// ___EM_Instance_9

// EM Instance DB
// EM_Instance_9
// DB726 = EM_Instance_9
// FB702 = EM_I_OUT
DATA_BLOCK DB726 FB702
BEGIN
END_DATA_BLOCK

FUNCTION "EM_Instance_9_FC" : VOID
TITLE =EM_Instance_9_FC
// EM_Instance_9_FC

AUTHOR :
FAMILY : 'eminst'
NAME : namehead
VERSION : 0.1

BEGIN

NETWORK
TITLE = Main
//--------------------------------
//
//--------------------------------

CALL EM_I_OUT, DB 726(
	em_id := 34,
	Pump_RUN := "M106".QNOFF2,
	PIC01_PV := "FIC101".PV,
	LT01_PV := "LT200".QfVal,
	BV_Bottom_OPN := "MV007".QOPEN,
	BV_Bottom_CLS := "MV007".QCLOSE,
	BV_Tran_M04_OPN := "MV003".QOPEN,
	BV_Tran_M04_CLS := "MV003".QCLOSE,
	Pump_ON := "M106".L_ON,
	PIC01_SP := "FIC101".HMI_SP_INT,
	PIC01_AUT := "FIC101".L_AUT,
	PIC01_VAL_OUT := "FIC101".HMI_MAN,
	PIC01_SET_SP := "FIC101".Set_SP,
	PIC01_SET_OUT := "FIC101".Set_Output,
	BV_Bottom_CMD := "MV007".AUT_OP,
	BV_Tran_M04_CMD := "MV003".AUT_OP
)



END_FUNCTION


// <SPLIT>EM_INSTANCE_EM_Instance_10.awl</SPLIT>


// ___EM_Instance_10

// EM Instance DB
// EM_Instance_10
// DB727 = EM_Instance_10
// FB702 = EM_I_OUT
DATA_BLOCK DB727 FB702
BEGIN
END_DATA_BLOCK

FUNCTION "EM_Instance_10_FC" : VOID
TITLE =EM_Instance_10_FC
// EM_Instance_10_FC

AUTHOR :
FAMILY : 'eminst'
NAME : namehead
VERSION : 0.1

BEGIN

NETWORK
TITLE = Main
//--------------------------------
//
//--------------------------------

CALL EM_I_OUT, DB 727(
	em_id := 35,
	Pump_RUN := "M106".QNOFF2,
	PIC01_PV := "FIC101".PV,
	LT01_PV := "LT101".QfVal,
	BV_Bottom_OPN := "MV007".QOPEN,
	BV_Bottom_CLS := "MV007".QCLOSE,
	Pump_ON := "M106".L_ON,
	PIC01_SP := "FIC101".HMI_SP_INT,
	PIC01_AUT := "FIC101".L_AUT,
	PIC01_VAL_OUT := "FIC101".HMI_MAN,
	PIC01_SET_SP := "FIC101".Set_SP,
	PIC01_SET_OUT := "FIC101".Set_Output,
	BV_Bottom_CMD := "MV007".AUT_OP
)



END_FUNCTION


// <SPLIT>EM_INSTANCE_EM_Instance_11.awl</SPLIT>


// ___EM_Instance_11

// EM Instance DB
// EM_Instance_11
// DB728 = EM_Instance_11
// FB702 = EM_I_OUT
DATA_BLOCK DB728 FB702
BEGIN
END_DATA_BLOCK

FUNCTION "EM_Instance_11_FC" : VOID
TITLE =EM_Instance_11_FC
// EM_Instance_11_FC

AUTHOR :
FAMILY : 'eminst'
NAME : namehead
VERSION : 0.1

BEGIN

NETWORK
TITLE = Main
//--------------------------------
//
//--------------------------------

CALL EM_I_OUT, DB 728(
	em_id := 36,
	Pump_RUN := "M106".QNOFF2,
	PIC01_PV := "FIC101".PV,
	LT01_PV := "LT201".QfVal,
	XV_Bottom_OPN := "XV001".QOPEN,
	XV_Bottom_CLS := "XV001".QCLOSE,
	Pump_ON := "M106".L_ON,
	PIC01_SP := "FIC101".HMI_SP_INT,
	PIC01_AUT := "FIC101".L_AUT,
	PIC01_VAL_OUT := "FIC101".HMI_MAN,
	PIC01_SET_SP := "FIC101".Set_SP,
	PIC01_SET_OUT := "FIC101".Set_Output,
	XV_Bottom_CMD := "XV001".AUT_OP
)



END_FUNCTION


// <SPLIT>EM_INSTANCE_EM_Instance_12.awl</SPLIT>


// ___EM_Instance_12

// EM Instance DB
// EM_Instance_12
// DB729 = EM_Instance_12
// FB702 = EM_I_OUT
DATA_BLOCK DB729 FB702
BEGIN
END_DATA_BLOCK

FUNCTION "EM_Instance_12_FC" : VOID
TITLE =EM_Instance_12_FC
// EM_Instance_12_FC

AUTHOR :
FAMILY : 'eminst'
NAME : namehead
VERSION : 0.1

BEGIN

NETWORK
TITLE = Main
//--------------------------------
//
//--------------------------------

CALL EM_I_OUT, DB 729(
	em_id := 37,
	Pump_RUN := "M106".QNOFF2,
	PIC01_PV := "FIC101".PV,
	LT01_PV := "LT201".QfVal,
	XV_Bottom_OPN := "XV002".QOPEN,
	XV_Bottom_CLS := "XV002".QCLOSE,
	Pump_ON := "M106".L_ON,
	PIC01_SP := "FIC101".HMI_SP_INT,
	PIC01_AUT := "FIC101".L_AUT,
	PIC01_VAL_OUT := "FIC101".HMI_MAN,
	PIC01_SET_SP := "FIC101".Set_SP,
	PIC01_SET_OUT := "FIC101".Set_Output,
	XV_Bottom_CMD := "XV002".AUT_OP
)



END_FUNCTION


// <SPLIT>EM_INSTANCE_EM_Instance_13.awl</SPLIT>


// ___EM_Instance_13

// EM Instance DB
// EM_Instance_13
// DB730 = EM_Instance_13
// FB702 = EM_I_OUT
DATA_BLOCK DB730 FB702
BEGIN
END_DATA_BLOCK

FUNCTION "EM_Instance_13_FC" : VOID
TITLE =EM_Instance_13_FC
// EM_Instance_13_FC

AUTHOR :
FAMILY : 'eminst'
NAME : namehead
VERSION : 0.1

BEGIN

NETWORK
TITLE = Main
//--------------------------------
//
//--------------------------------

CALL EM_I_OUT, DB 730(
	em_id := 38,
	Pump_RUN := "M106".QNOFF2,
	PIC01_PV := "FIC101".PV,
	LT01_PV := "LT201".QfVal,
	XV_Bottom_OPN := "XV003".QOPEN,
	XV_Bottom_CLS := "XV003".QCLOSE,
	Pump_ON := "M106".L_ON,
	PIC01_SP := "FIC101".HMI_SP_INT,
	PIC01_AUT := "FIC101".L_AUT,
	PIC01_VAL_OUT := "FIC101".HMI_MAN,
	PIC01_SET_SP := "FIC101".Set_SP,
	PIC01_SET_OUT := "FIC101".Set_Output,
	XV_Bottom_CMD := "XV003".AUT_OP
)



END_FUNCTION


// <SPLIT>EM_INSTANCE_EM_Instance_14.awl</SPLIT>


// ___EM_Instance_14

// EM Instance DB
// EM_Instance_14
// DB731 = EM_Instance_14
// FB702 = EM_I_OUT
DATA_BLOCK DB731 FB702
BEGIN
END_DATA_BLOCK

FUNCTION "EM_Instance_14_FC" : VOID
TITLE =EM_Instance_14_FC
// EM_Instance_14_FC

AUTHOR :
FAMILY : 'eminst'
NAME : namehead
VERSION : 0.1

BEGIN

NETWORK
TITLE = Main
//--------------------------------
//
//--------------------------------

CALL EM_I_OUT, DB 731(
	em_id := 39,
	Pump_RUN := "M106".QNOFF2,
	PIC01_PV := "FIC101".PV,
	LT01_PV := "LT201".QfVal,
	XV_Bottom_OPN := "XV004".QOPEN,
	XV_Bottom_CLS := "XV004".QCLOSE,
	Pump_ON := "M106".L_ON,
	PIC01_SP := "FIC101".HMI_SP_INT,
	PIC01_AUT := "FIC101".L_AUT,
	PIC01_VAL_OUT := "FIC101".HMI_MAN,
	PIC01_SET_SP := "FIC101".Set_SP,
	PIC01_SET_OUT := "FIC101".Set_Output,
	XV_Bottom_CMD := "XV004".AUT_OP
)



END_FUNCTION



// <SPLIT>PHASE_INSTANCE_phase_1.awl</SPLIT>


// ___phase_1

// Phase Instance DB
// DB716 = phase_1
// FB701 = phase_example
DATA_BLOCK DB716 FB701
BEGIN
END_DATA_BLOCK

FUNCTION "phase_1_FC" : VOID
TITLE =phase_1_FC
// phase_1_FC
// First instance of fds_example
AUTHOR :
FAMILY : 'phseinst'
NAME : namehead
VERSION : 0.1

BEGIN
NETWORK
TITLE = Main
//--------------------------------
// Call the phase
//--------------------------------

CALL phase_example, DB 716
	(XV003_OPN := "XV300".QOPEN,
	XV004_OPN := "XV400".QOPEN,
	XV005_OPN := "XV500".QOPEN,
	P001_RUN := "P100".QRUN,
	LT001_PV := "LT100".QfVal,
	LT002_PV := "LT200".QfVal,
	XV003_CMD := "XV300".AUT_OP,
	XV004_CMD := "XV400".AUT_OP,
	P001_ON := "P100".AUTO_ON,
	FIC001_EXT := "FIC100".L_REMOTE,
	FIC001_SP := "FIC100".HMI_SP_INT,
	FIC001_AUT := "FIC100".L_AUT,
	FIC001_VAL_OUT := "FIC100".HMI_MAN,
	FIC001_SET_SP := "FIC100".Set_SP,
	FIC001_SET_OUT := "FIC100".Set_Output);



END_FUNCTION


// <SPLIT>PHASE_INSTANCE_phase_2.awl</SPLIT>


// ___phase_2

// Phase Instance DB
// DB717 = phase_2
// FB701 = phase_example
DATA_BLOCK DB717 FB701
BEGIN
END_DATA_BLOCK

FUNCTION "phase_2_FC" : VOID
TITLE =phase_2_FC
// phase_2_FC
// Second instance of fds_example
AUTHOR :
FAMILY : 'phseinst'
NAME : namehead
VERSION : 0.1

BEGIN
NETWORK
TITLE = Main
//--------------------------------
// Call the phase
//--------------------------------

CALL phase_example, DB 717
	(XV003_OPN := "XV301".QOPEN,
	XV004_OPN := "XV401".QOPEN,
	XV005_OPN := "XV501".QOPEN,
	P001_RUN := "P101".QRUN,
	LT001_PV := "LT101".QfVal,
	LT002_PV := "LT201".QfVal,
	XV003_CMD := "XV301".AUT_OP,
	XV004_CMD := "XV401".AUT_OP,
	P001_ON := "P101".AUTO_ON,
	FIC001_EXT := "FIC101".L_REMOTE,
	FIC001_SP := "FIC101".HMI_SP_INT,
	FIC001_AUT := "FIC101".L_AUT,
	FIC001_VAL_OUT := "FIC101".HMI_MAN,
	FIC001_SET_SP := "FIC101".Set_SP,
	FIC001_SET_OUT := "FIC101".Set_Output);



END_FUNCTION


// <SPLIT>main_program.awl</SPLIT>

// ___Control_Modules
FUNCTION Control_Modules : VOID
TITLE = Control_Modules
// Call all the Control Modules
AUTHOR:
FAMILY: 'program'
NAME: namehead
VERSION: 0.1

BEGIN

NETWORK
TITLE =
//--------------------------------
//
//--------------------------------
	CALL	XV001_FC;
	CALL	XV002_FC;
	CALL	XV003_FC;
	CALL	XV004_FC;
	CALL	XV300_FC;
	CALL	XV400_FC;
	CALL	XV500_FC;
	CALL	XV301_FC;
	CALL	XV501_FC;
	CALL	XV401_FC;
	CALL	MV001_FC;
	CALL	MV002_FC;
	CALL	MV003_FC;
	CALL	MV004_FC;
	CALL	MV005_FC;
	CALL	MV006_FC;
	CALL	MV007_FC;
	CALL	P100_FC;
	CALL	P200_FC;
	CALL	P101_FC;
	CALL	P201_FC;
	CALL	M100_FC;
	CALL	M101_FC;
	CALL	M102_FC;
	CALL	M103_FC;
	CALL	M104_FC;
	CALL	M105_FC;
	CALL	M106_FC;
	CALL	LT001_FC;
	CALL	LT002_FC;
	CALL	LT003_FC;
	CALL	LT004_FC;
	CALL	LT005_FC;
	CALL	LT006_FC;
	CALL	LT007_FC;
	CALL	LT100_FC;
	CALL	LT200_FC;
	CALL	LT101_FC;
	CALL	LT201_FC;
	CALL	LS001_FC;
	CALL	LS002_FC;
	CALL	LIC001_FC;
	CALL	LIC002_FC;
	CALL	LIC003_FC;
	CALL	LIC004_FC;
	CALL	LIC005_FC;
	CALL	LIC006_FC;
	CALL	FIC100_FC;
	CALL	FIC101_FC;

END_FUNCTION

// ___Equipment_Modules
FUNCTION Equipment_Modules : VOID
TITLE = Equipment_Modules
// Call all the Equipment Modules
AUTHOR:
FAMILY: 'program'
NAME: namehead
VERSION: 0.1

BEGIN

NETWORK
TITLE =
//--------------------------------
//
//--------------------------------
	CALL	EM_Instance_1_FC;
	CALL	EM_Instance_2_FC;
	CALL	EM_Instance_3_FC;
	CALL	EM_Instance_4_FC;
	CALL	EM_Instance_5_FC;
	CALL	EM_Instance_6_FC;
	CALL	EM_Instance_7_FC;
	CALL	EM_Instance_8_FC;
	CALL	EM_Instance_9_FC;
	CALL	EM_Instance_10_FC;
	CALL	EM_Instance_11_FC;
	CALL	EM_Instance_12_FC;
	CALL	EM_Instance_13_FC;
	CALL	EM_Instance_14_FC;

END_FUNCTION

// ___Phases
FUNCTION Phases : VOID
TITLE = Phases
// Call all the Phases
AUTHOR:
FAMILY: 'program'
NAME: namehead
VERSION: 0.1

BEGIN

NETWORK
TITLE =
//--------------------------------
//
//--------------------------------
	CALL	phase_1_FC;
	CALL	phase_2_FC;

END_FUNCTION

// ___Units
FUNCTION Units : VOID
TITLE = Units
// Call all the Units
AUTHOR:
FAMILY: 'program'
NAME: namehead
VERSION: 0.1

BEGIN

NETWORK
TITLE =
//--------------------------------
//
//--------------------------------

END_FUNCTION

// ___Main_Program
FUNCTION Main_Program : VOID
TITLE = Main_Program
// Call all the program components
AUTHOR:
FAMILY: 'program'
NAME: namehead
VERSION: 0.1

BEGIN

NETWORK
TITLE =
//--------------------------------
//
//--------------------------------

	CALL	Control_Modules;
	CALL	Equipment_Modules;
	CALL	Phases;
	CALL	Units;

END_FUNCTION

// ___OB1
// OB1 only calls Main_Program
// Comment this whole section if some code needs to be entered manually
// => in this case make another program structure starting from OB1
ORGANIZATION_BLOCK OB 1
TITLE = "Main Program Sweep (Cycle)"
VERSION : 0.1


VAR_TEMP
  OB1_EV_CLASS : BYTE ;	//Bits 0-3 = 1 (Coming event), Bits 4-7 = 1 (Event class 1)
  OB1_SCAN_1 : BYTE ;	//1 (Cold restart scan 1 of OB 1), 3 (Scan 2-n of OB 1)
  OB1_PRIORITY : BYTE ;	//Priority of OB Execution
  OB1_OB_NUMBR : BYTE ;	//1 (Organization block 1, OB1)
  OB1_RESERVED_1 : BYTE ;	//Reserved for system
  OB1_RESERVED_2 : BYTE ;	//Reserved for system
  OB1_PREV_CYCLE : INT ;	//Cycle time of previous OB1 scan (milliseconds)
  OB1_MIN_CYCLE : INT ;	//Minimum cycle time of OB1 (milliseconds)
  OB1_MAX_CYCLE : INT ;	//Maximum cycle time of OB1 (milliseconds)
  OB1_DATE_TIME : DATE_AND_TIME ;	//Date and time OB1 started
END_VAR
BEGIN

NETWORK
TITLE =
//--------------------------------
//
//--------------------------------

	CALL	Main_Program;

END_ORGANIZATION_BLOCK







